{attribute 'call_after_init'}
FUNCTION_BLOCK FB_AxisParametersNC IMPLEMENTS I_AxisParameters
VAR_INPUT
END_VAR
VAR_OUTPUT
END_VAR
VAR
    {attribute 'no_copy'}
    AxisRef : REFERENCE TO AXIS_REF;
    iPersistentDataStorage : I_PersistentDataStorage;

    nRawEncoderULINT AT %I*: ULINT;
    // Raw encoder IO for UINT (Relative Encoders)
    nRawEncoderUINT AT %I*: UINT;
    // Raw encoder IO for INT (LVDT)
    nRawEncoderINT AT %I*: INT;
    // Raw encoder IO for INT (EL5072 LVDT)
    nRawEncoderDINT AT %I*: DINT;
    // Encoder count summary, if linked above
    {attribute 'pytmc' := '
        pv: PLC:nEncoderCount
        io: i
        field: DESC Count from encoder hardware
    '}
    nEncoderCount: UDINT;
    // Position lag difference
    {attribute 'pytmc' := '
        pv: PLC:fPosDiff
        io: i
        field: DESC Position lag difference
    '}
    fPosDiff: LREAL;
    // NC parameters that are exposed with pytmc pragmas
    {attribute 'pytmc' := '
        pv: PLC:AxisPar
        io: i
        field: DESC Axis configuration parameters in the numerical controller.
    '}
    stAxisParametersExposed : ST_AxisParameterSetExposed;
    // MC_ReadParameterSet Output
    mcReadParams: MC_ReadParameterSet;
    //{attribute 'hide'}
    stAxisParameters: ST_AxisParameterSet;
    bNcParamsReadInit   : BOOL;
    // save and restore
    fbSetPos: MC_SetPosition;
    bClearPositionLag : BOOL := TRUE;
    NCParamsTimer : TON;
    bAxisParamsInit : BOOL;
    nLatchErrId : BOOL;
    bRestoreDone 	: BOOL;
    bRestoreError 	: BOOL;
    nRestoreErrorID : UDINT;
    // save and Restore
    RestoreTimer: TON;
    bRestoreInit: BOOL;
    bRestoreLoad: BOOL;
    nLatchError: UDINT;
    bEncError: BOOL;
    tRetryDelay: TIME := T#1S;
    tRefreshDelay: TIME := T#1S;
    bUpdateEnable : BOOL;
    bExecute : BOOL;
    nMaxRetries: UINT := 10;
    nCurrTries: UINT := 0;
    bRestoreWaitRetry: BOOL;
    tonRestoreRetry: TON;
    tRefreshTime : TIME := T#1S;
    bError				: BOOL;
    nErrorId			: UDINT:=0;
    sMessage : T_MAXSTRING;

    bSaveEnabled	: BOOL := TRUE;
    bDone : BOOL;
    bBusy    : BOOL;
END_VAR

VAR PERSISTENT
    {attribute 'conditionalshow'}
    bSaved: BOOL;
    {attribute 'conditionalshow'}
    fSavedPosition: LREAL;
END_VAR

THIS^.AxisRef.ReadStatus();

// Calibrate raw encoder data
THIS^.ScaleRawEncoder();

// Periodic update of NC parameters
NCParamsTimer( IN:=bUpdateEnable AND NOT bExecute, PT:=tRefreshDelay);
bExecute S= NCParamsTimer.Q;
mcReadParams(
    Parameter:=THIS^.stAxisParameters,
    Axis:=THIS^.AxisRef,
    Execute:=bUpdateEnable AND bExecute,
    Error=>bError,
    ErrorID=>nErrorID,
    Busy=>bBusy,
    Done => bDone);

// Copy axis parameters that we want to expose to the EPICS layer.
THIS^.stAxisParametersExposed.bCtrlEnablePosDiffControl     := THIS^.stAxisParameters.bCtrlEnablePosDiffControl;
THIS^.stAxisParametersExposed.bEncEnableSoftEndMaxControl   := THIS^.stAxisParameters.bEncEnableSoftEndMaxControl;
THIS^.stAxisParametersExposed.bEncEnableSoftEndMinControl   := THIS^.stAxisParameters.bEncEnableSoftEndMinControl;
THIS^.stAxisParametersExposed.fAccelerationMax              := THIS^.stAxisParameters.fAccelerationMax;
THIS^.stAxisParametersExposed.fCtrlPosDiffMax               := THIS^.stAxisParameters.fCtrlPosDiffMax;
THIS^.stAxisParametersExposed.fCtrlPosDiffMaxTime           := THIS^.stAxisParameters.fCtrlPosDiffMaxTime;
THIS^.stAxisParametersExposed.fDecelerationMax              := THIS^.stAxisParameters.fDecelerationMax;
THIS^.stAxisParametersExposed.fEncSoftEndMax                := THIS^.stAxisParameters.fEncSoftEndMax;
THIS^.stAxisParametersExposed.fEncSoftEndMin                := THIS^.stAxisParameters.fEncSoftEndMin;
THIS^.stAxisParametersExposed.fVeloMaximum                  := THIS^.stAxisParameters.fVeloMaximum;
THIS^.stAxisParametersExposed.fEncOffset               		:= THIS^.stAxisParameters.fEncOffset;
THIS^.stAxisParametersExposed.fEncScaleFactorInternal       := THIS^.stAxisParameters.fEncScaleFactorInternal;

IF mcReadParams.ErrorID <> 0 THEN
    nLatchErrId := 0;
END_IF
bExecute R= mcReadParams.Done OR mcReadParams.Error;
THIS^.bAxisParamsInit S= mcReadParams.Done;


// Save Encoder position
// needs some pre-conditions to use persistent storage
IF bSaveEnabled THEN
    // Check ST_MotionStage for an encoder error (range 0x44nn)
    bEncError:= AxisRef.Status.Error AND  ( AxisRef.Status.ErrorID  >= 16#4400  AND AxisRef.Status.ErrorID <= 16#44FF );
    // Do not save if we're currently loading or if there is an encoder error
    IF NOT bRestoreLoad AND NOT bEncError AND NOT bRestoreWaitRetry THEN
        fSavedPosition := AxisRef.NcToPlc.ActPos;
        // This persistent variable lets us check if anything was saved
        // It will be TRUE at startup if we have saved values
        bSaved := TRUE;
        (*
            use this with a timer of a change threshold on the fActPosition
            to trigger a save from this PLC program. otherwise this will be a spamming
            persistence, filling up the disk.
        *)
        //iPersistentDataStorage.TriggerWriteOfPersistentData := bSaveEnabled;
    END_IF
END_IF

{warning 'Add property implementation'}
PROPERTY Aborted : BOOL
GET
END_GET
END_PROPERTY

{warning 'Add property implementation'}
PROPERTY Active : BOOL
GET
END_GET
END_PROPERTY

{warning 'add property implementation'}
PROPERTY AxisParamsInit : BOOL
GET
AxisParamsInit := bAxisParamsInit;
END_GET
END_PROPERTY

{warning 'Add property implementation'}
PROPERTY Busy : BOOL
GET
END_GET
END_PROPERTY

{warning 'Add property implementation'}
PROPERTY Done : BOOL
GET
END_GET
END_PROPERTY

METHOD EncoderParamsSave
VAR_INPUT
    Enable	: BOOL;
END_VAR
THIS^.bSaveEnabled := Enable;
END_METHOD

{warning 'add property implementation'}
PROPERTY Error : BOOL
GET
Error := bError;
END_GET
END_PROPERTY

{warning 'add property implementation'}
PROPERTY ErrorID : UDINT
GET
ErrorID := nErrorID;
END_GET
END_PROPERTY

METHOD ExposeAxisParams
VAR_INPUT
    Enable: BOOL;
    RefreshDelay: TIME;
END_VAR
THIS^.bUpdateEnable:= Enable;
THIS^.tRefreshDelay:= RefreshDelay;
END_METHOD

//FB_Init is always available implicitly and it is used primarily for initialization.
//The return value is not evaluated. For a specific influence, you can also declare the
//methods explicitly and provide additional code there with the standard initialization
//code. You can evaluate the return value.
METHOD FB_Init: BOOL
VAR_INPUT
    bInitRetains: BOOL; // TRUE: the retain variables are initialized (reset warm / reset cold)
    bInCopyCode: BOOL;  // TRUE: the instance will be copied to the copy code afterward (online change)
    AxisRef : REFERENCE TO AXIS_REF;
    iPersistentDataStorage : I_PersistentDataStorage;
END_VAR
THIS^.AxisRef REF= AxisRef;
THIS^.iPersistentDataStorage := iPersistentDataStorage;
END_METHOD

PROPERTY Message : T_MAXSTRING
GET
Message := sMessage;
END_GET
END_PROPERTY

{warning 'add property implementation'}
PROPERTY RefVeloSearch : LREAL
GET
RefVeloSearch := THIS^.stAxisParameters.fRefVeloSearch;
END_GET
END_PROPERTY

{warning 'add property implementation'}
PROPERTY RefVeloSync : LREAL
GET
RefVeloSync:= THIS^.stAxisParameters.fRefVeloSync;
END_GET
END_PROPERTY

{attribute 'call_after_init'}
METHOD RestoreAxisParams
// Trigger a load if anything was saved at all
IF NOT bRestoreInit THEN
    bRestoreInit := TRUE;
    bRestoreLoad S= bSaved;
    fbSetPos.Options.ClearPositionLag := TRUE;
END_IF

// Set our position if bRestoreLoad is true
fbSetPos( Axis:=THIS^.AxisRef, Execute:=bRestoreLoad, Position:=fSavedPosition);

// Only load once, at startup
bRestoreLoad R= fbSetPos.Done OR fbSetPos.Error;

IF fbSetPos.Error THEN
    // Keep the error latched, it can disappear if Execute is set to FALSE
    nLatchError := fbSetPos.ErrorID;
    nCurrTries := nCurrTries + 1;
    IF nCurrTries >= nMaxRetries THEN
    // Alert the user that something has gone wrong
    bError := TRUE;
        nErrorId := nLatchError;
        sMessage := 'Error loading previously saved position.';
    ELSE
        // Reset the FB for the next retry
        fbSetPos( Axis:=THIS^.AxisRef, Execute:=bRestoreLoad, Position:=fSavedPosition);
        // Try again
        bRestoreWaitRetry := TRUE;
    END_IF
ELSE
    THIS^.bRestoreDone := TRUE;
END_IF

tonRestoreRetry( IN := bRestoreWaitRetry, PT := tRetryDelay);
bRestoreLoad S= tonRestoreRetry.Q;
bRestoreWaitRetry R= tonRestoreRetry.Q;
END_METHOD

{warning 'add property implementation'}
PROPERTY RestoreDone : BOOL
GET
END_GET
END_PROPERTY

{warning 'add property implementation'}
PROPERTY SavedPosition : LREAL
GET
SavedPosition := fSavedPosition;
END_GET
END_PROPERTY

{warning 'add property implementation'}
PROPERTY ScaledEncoderCount : UDINT
GET
END_GET
END_PROPERTY

METHOD ScaleRawEncoder : UDINT
IF nRawEncoderULINT <> 0 THEN
    IF nRawEncoderULINT < 4294967296 THEN
        nEncoderCount := ULINT_TO_UDINT(nRawEncoderULINT);
    ELSE
        nEncoderCount := ULINT_TO_UDINT(18446744073709551615 - nRawEncoderULINT);
    END_IF
ELSIF nRawEncoderUINT <> 0 THEN
    nEncoderCount := UINT_TO_UDINT(nRawEncoderUINT);
ELSIF nRawEncoderINT <> 0 THEN
    nEncoderCount := INT_TO_UDINT(nRawEncoderINT);
ELSIF nRawEncoderDINT <> 0 THEN
    nEncoderCount := DINT_TO_UDINT(nRawEncoderDINT);
ELSE
    nEncoderCount := 0;
END_IF

ScaleRawEncoder := nEncoderCount ;
END_METHOD

END_FUNCTION_BLOCK

(* stored: Version 1.1.0.1
   POU FB_AxisParametersNC: Id {7f8d36cc-18a1-4d6c-99dd-bd0795394dcd}, SpecialFunc None
   Property Aborted: Id {6f730b0b-0a56-4d4b-b10c-7aa6d451ffb9}
   Get Get: Id {195d6a7f-01a2-451b-aa25-a64fd76e79b7}
   Property Active: Id {b22df6f2-a22f-4a34-ae94-cfb631a24757}
   Get Get: Id {d1a9a3ed-fe85-4bb0-87cf-89cdb316a968}
   Property AxisParamsInit: Id {a0575603-f379-443c-8fcf-402542f903ce}
   Get Get: Id {2ef7b70d-e8b5-4a7c-b6d9-8882f4c8d790}
   Property Busy: Id {e5dec030-d598-46fd-afca-22fd9bde3a46}
   Get Get: Id {51885e31-af8a-4a94-a215-169272d4b781}
   Property Done: Id {a3a56a42-9da7-40a8-925f-55df107c55cd}
   Get Get: Id {ec9b7af9-7f82-4fed-872e-fdb89505987f}
   Method EncoderParamsSave: Id {29eaeb35-c218-4604-adff-fca8f06a68eb}
   Property Error: Id {239ac2b3-3c2a-4399-a932-e6c718d2e1bb}
   Get Get: Id {4e85ac84-f8ba-45e9-84c6-7c5588481cb5}
   Property ErrorID: Id {7fc4dd77-9990-47fb-a3f3-15f5d1c36a93}
   Get Get: Id {d39cb682-a948-4eed-b151-61c04c28fc87}
   Method ExposeAxisParams: Id {d1c3b848-a85c-4697-aa4e-a392a6f23769}
   Method FB_Init: Id {6c116c09-ef45-432c-8e07-3fe37fad5966}
   Property Message: Id {32b322a0-2932-4424-b95e-453b6c119c35}
   Get Get: Id {e135d05b-80a3-4ab1-9f4a-39e3dfbcfa43}
   Property RefVeloSearch: Id {5735fb85-0be0-4a0c-80a8-b61350b0c2d1}
   Get Get: Id {af40d57e-8351-45be-9af1-5d364693fb2b}
   Property RefVeloSync: Id {a6e12d44-9094-4586-b6c6-065562b64be3}
   Get Get: Id {dfa185c9-0e75-4040-80b1-2e94d9447652}
   Method RestoreAxisParams: Id {68aa741c-8d0b-49b0-a5c7-e5cb1bf9c532}
   Property RestoreDone: Id {e7e6ffa0-ec40-4879-b319-9d4ca78e63b6}
   Get Get: Id {4baad02a-e870-46d0-aa29-7a3586bea07c}
   Property SavedPosition: Id {4a2e7fd2-dff9-49f3-8bb0-6e6d2bbd5bd1}
   Get Get: Id {47036862-e42a-472d-9c02-661c5f9aa886}
   Property ScaledEncoderCount: Id {d81c0e55-4ea7-4a05-869f-d72e8a4ea95e}
   Get Get: Id {3c473915-1f59-45dd-90cc-be2e45b56ba4}
   Method ScaleRawEncoder: Id {eb3341cc-367a-44d0-8a42-35c37667da1b} *)
